// TIA Portal V18 export
TYPE "LGasp_TypeERP"
// stored: IsFailsafeCompliant false
   STRUCT
      eventlog_PLC_PC_bool { ExternalAccessible := 'False'; ExternalVisible := 'False'; ExternalWritable := 'False'} : Array[1..32] of Bool;
      eventlog_PLC_PC : DWord;
      eventlog_PC_PLC : Array[1..32] of Bool;
      dati_PLC_PC : "LGasp_TypeData_toERP";
      dati_PC_PLC : "LGasp_TypeData_fromERP";
   END_STRUCT;
   // // eventlog_PLC_PC_bool[1] : FP_emergenza
   // // eventlog_PLC_PC_bool[2] : FN_emergenza
   // // eventlog_PLC_PC_bool[3] : FP_manuale
   // // eventlog_PLC_PC_bool[4] : FN_manuale
   // // eventlog_PLC_PC_bool[5] : FP_semiautomatico
   // // eventlog_PLC_PC_bool[6] : FN_semiautomatico
   // // eventlog_PLC_PC_bool[7] : FP_automatico
   // // eventlog_PLC_PC_bool[8] : FN_automatico
   // // eventlog_PLC_PC_bool[9] : marcia_macchina
   // // eventlog_PLC_PC_bool[10] : arresto_macchina
   // // eventlog_PLC_PC_bool[11] : inizio_ODL
   // // eventlog_PLC_PC_bool[12] : fIne_ODL
   // // eventlog_PLC_PC_bool[13] : fIne_pacco
   // // eventlog_PLC_PC_bool[14] : arresto_macchina_da_pulsante
   // // eventlog_PLC_PC_bool[15] : pezzo_tagliato
   // // eventlog_PLC_PC_bool[16] : articolo_terminato
   // // eventlog_PLC_PC_bool[17] : profila in marcia
   // // eventlog_PLC_PC_bool[18] : profila ferma
   // // eventlog_PLC_PC_bool[19] : pezzo tagliato scarto
   // // eventlog_PLC_PC_bool[20] : bool_19
   // // eventlog_PLC_PC_bool[21] : bool_20
   // // eventlog_PLC_PC_bool[22] : bool_21
   // // eventlog_PLC_PC_bool[23] : bool_22
   // // eventlog_PLC_PC_bool[24] : bool_23
   // // eventlog_PLC_PC_bool[25] : bool_24
   // // eventlog_PLC_PC_bool[26] : bool_25
   // // eventlog_PLC_PC_bool[27] : bool_26
   // // eventlog_PLC_PC_bool[28] : bool_27
   // // eventlog_PLC_PC_bool[29] : bool_28
   // // eventlog_PLC_PC_bool[30] : bool_29
   // // eventlog_PLC_PC_bool[31] : bool_30
   // // eventlog_PLC_PC_bool[32] : bool_31
   // // eventlog_PC_PLC[1] : FP_emergenza
   // // eventlog_PC_PLC[2] : FN_emergenza
   // // eventlog_PC_PLC[3] : FP_manuale
   // // eventlog_PC_PLC[4] : FN_manuale
   // // eventlog_PC_PLC[5] : FP_semiautomatico
   // // eventlog_PC_PLC[6] : FN_semiautomatico
   // // eventlog_PC_PLC[7] : FP_automatico
   // // eventlog_PC_PLC[8] : FN_automatico
   // // eventlog_PC_PLC[9] : marcia_macchina
   // // eventlog_PC_PLC[10] : arresto_macchina
   // // eventlog_PC_PLC[11] : inizio_ODL
   // // eventlog_PC_PLC[12] : fIne_ODL
   // // eventlog_PC_PLC[13] : fIne_pacco
   // // eventlog_PC_PLC[14] : arresto_macchina_da_pulsante
   // // eventlog_PC_PLC[15] : pezzo_tagliato
   // // eventlog_PC_PLC[16] : articolo_terminato
   // // eventlog_PC_PLC[17] : profila in marcia
   // // eventlog_PC_PLC[18] : profila ferma
   // // eventlog_PC_PLC[19] : pezzo tagliato scarto
   // // eventlog_PC_PLC[20] : bool_19
   // // eventlog_PC_PLC[21] : bool_20
   // // eventlog_PC_PLC[22] : bool_21
   // // eventlog_PC_PLC[23] : bool_22
   // // eventlog_PC_PLC[24] : bool_23
   // // eventlog_PC_PLC[25] : bool_24
   // // eventlog_PC_PLC[26] : bool_25
   // // eventlog_PC_PLC[27] : bool_26
   // // eventlog_PC_PLC[28] : bool_27
   // // eventlog_PC_PLC[29] : bool_28
   // // eventlog_PC_PLC[30] : bool_29
   // // eventlog_PC_PLC[31] : bool_30
   // // eventlog_PC_PLC[32] : bool_31
END_TYPE
